FUNCTION_BLOCK MOD_OccupationIds (* OPC UA and local channel IDs of the occupation *)
  (* Standard: 61499-2 *)
  (* Version 0.1, 2026-09-28, Project contributors, AAU Smart Production Lab *)
  PACKAGE modlib;
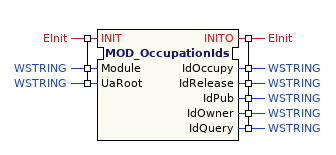
  EVENT_INPUT
    INIT : EInit WITH Module, UaRoot;
  END_EVENT
  EVENT_OUTPUT
    INITO : EInit WITH IdOccupy, IdRelease, IdPub, IdOwner, IdQuery;
  END_EVENT
  VAR_INPUT
    Module : WSTRING;
    UaRoot : WSTRING;
  END_VAR
  VAR_OUTPUT
    IdOccupy : WSTRING;
    IdRelease : WSTRING;
    IdPub : WSTRING;
    IdOwner : WSTRING;
    IdQuery : WSTRING;
  END_VAR
  EC_STATES
    INIT : INIT -> INITO;
  END_STATES
  ALGORITHM INIT IN ST:
IdOccupy := CONCAT(CONCAT(CONCAT("opc_ua[CREATE_METHOD;", CONCAT(UaRoot, "/Occupation/")), "Occupy"), "]");
IdRelease := CONCAT(CONCAT(CONCAT("opc_ua[CREATE_METHOD;", CONCAT(UaRoot, "/Occupation/")), "Release"), "]");
IdPub := CONCAT(CONCAT(CONCAT("opc_ua[WRITE;", CONCAT(UaRoot, "/Occupation/")), "Occupied"), "]");
IdOwner := CONCAT(CONCAT("loc[", Module), "/owner]");
IdQuery := CONCAT(CONCAT("loc[", Module), "/owner/query]");
  END_ALGORITHM
END_FUNCTION_BLOCK
